FUNCTION_BLOCK FB_GameSetup
VAR_INPUT
END_VAR
VAR_OUTPUT
END_VAR
VAR
	i	: DINT;
	j	: DINT;
	k	: DINT;
	m	: INT;
END_VAR

// Decode sequencer step bits
MEMSET(ADR(GVL_Global.bStep), 0, SIZEOF(GVL_Global.bStep));
GVL_Global.stGameSetup.stStep[GVL_Global.stGameSetup.iStepNumber] := TRUE;

//Choose blackjack variation: 1 - Common BlackJack, 2 - Free Bet BlackJack, 3 - Spanish 21
IF GVL_Global.eBJVariation.Idle = GVL_Global.iVariationSelection THEN
	//Wait for user to select a BlackJack variation
	GVL_Global.sInstruction := 'Please choose a blackjack variation to play.';
END_IF

IF GVL_Global.iVariationSelection >= 1 AND GVL_Global.iVariationSelection <= 3 THEN
	//Set up initial information regarding card, card suit, and deck information
	FOR m := 0 TO 9 DO
		GVL_Global.stGameSetup.sCards[m] := INT_TO_STRING(m+2);
	END_FOR
	GVL_Global.stGameSetup.sCards[10] := 'J';
	GVL_Global.stGameSetup.sCards[11] := 'Q';
	GVL_Global.stGameSetup.sCards[12] := 'K';
	GVL_Global.stGameSetup.sCards[13] := 'A';
	
	GVL_Global.stGameSetup.sCardSuit[0] := 'Clubs';
	GVL_Global.stGameSetup.sCardSuit[1] := 'Diamonds';
	GVL_Global.stGameSetup.sCardSuit[2] := 'Bishops';
	GVL_Global.stGameSetup.sCardSuit[3] := 'Hearts';
	GVL_Global.stGameSetup.iStepNumber := 2;
ELSE
	GVL_Global.stGameSetup.iStepNumber := 0;
END_IF

//GVL_Global.sInstruction := 'Please choose a blackjack variation to play.';
//IF GVL_Global.iVariationSelection >=1 AND GVL_Global.iVariationSelection <= 3 THEN
//	GVL_Global.stGameSetup.iStepNumber := 2;
//ELSE
//	GVL_Global.stGameSetup.iStepNumber := 0;
//END_IF

//Error State
IF GVL_Global.stGameSetup.stStep.bStep[0] THEN
	//False entry was entered
	GVL_Global.stGamePlay.sMessageType.sErrorMessage := 'You entered a wrong variation input. Please try again.';
	GVL_Global.stGamePlay.bVariationSelected := FALSE;
	GVL_Global.stGamePlay.iVariationSelection := 0;
END_IF


//Idle State
IF GVL_Global.stGameSetup.stStep.bStep[1] THEN
	GVL_Global.stGamePlay.sMessageType.sErrorMessage := 'Game is ongoing.';
	IF GVL_Global.stGamePlay.bReadyToStart AND GVL_Global.stGameSetup.bBankRollComplete THEN
		GVL_Global.stGamePlay.iStepNumber := 1;
	ELSE
		GVL_Global.stGamePlay.iStepNumber := 0;
	END_IF
END_IF

//Blackjack Deviation Selection
IF GVL_Global.stGameSetup.stStep.bStep[2] THEN
	IF GVL_Global.eBJVariation.Common_BlackJack = GVL_Global.iVariationSelection THEN
		//Common Blackjack was selected
		GVL_Global.stGameSetup.stMessageType.sInstructionMessage := 'Variation selected: Common Blackjack.';
	ELSIF GVL_Global.eBJVariation.FreeBet_BlackJack = GVL_Global.iVariationSelection THEN
		GVL_Global.stGameSetup.stMessageType.sInstructionMessage := 'Variation selected: Free Bet Blackjack.';
	ELSIF GVL_Global.eBJVariation.Spanish21 = GVL_Global.iVariationSelection THEN
		GVL_Global.stGameSetup.stMessageType.sInstructionMessage := 'Variation selected: Spanish 21.';
	END_IF
	GVL_Global.stGameSetup.iStepNumber := 3;
END_IF

//Choose 2 sidebets: 1 - Buster BlackJack, 2 - Dealer 16, 3 - Lucky Lucky, 4 - Match the Dealer, 5 - Pot of Gold (TBD)
//Side Bets Selection
IF GVL_Global.stGameSetup.stStep.bStep[3] THEN
	GVL_Global.stGameSetup.stMessageType.sRulesForGame[0] := 'Choose two (2) side bets: 1 - Buster BlackJack, 2 - Dealer 16, 3 - Lucky Lucky, 4 - Match the Dealer, 5 - Pot of Gold';
	GVL_Global.stGameSetup.stMessageType.sInstructionMessage[1] := 'Enter in text box labeled -> Side Bets To Play';
	GVL_Global.stGameSetup.stMessageType.sInstructionMessage[2] := 'Choose two (2) side bets: 1 - Buster BlackJack, 2 - Dealer 16, 3 - Lucky Lucky, 4 - Match the Dealer, 5 - Pot of Gold';
	GVL_Global.stGameSetup.stMessageType.sInstructionMessage := 'Enter in the following prompt: #,#';
	//Side Bet Choices Decoded
	GVL_Global.stGameSetup.stSideBetChoice.iFind := FIND(',',GVL_Global.stGameSetup.stSideBetChoice.sSideBetSelections);
	GVL_Global.stGameSetup.stSideBetChoice.iSideBet_One := STRING_TO_INT(LEFT(GVL_Global.stGameSetup.stSideBetChoice.sSideBetSelections,GVL_Global.stGameSetup.stSideBetChoice.iFind-1));
	GVL_Global.stGameSetup.stSideBetChoice.iSideBet_Two := STRING_TO_INT(RIGHT(GVL_Global.stGameSetup.stSideBetChoice.sSideBetSelections,GVL_Global.stGameSetup.stSideBetChoice.iFind+1));
	//Side bet #1 chosen
	IF GVL_Global.stGameSetup.stSideBetChoice.iSideBet_One = GVL_Global.stGameSetup.stSideBetChoice.eSideBetChoice.BusterBlackjack THEN
		GVL_Global.stGameSetup.stSideBetChoice.bBusterBlackjackSelected := TRUE;
		//GVL_Global.stGameSetup.sSideBetChoice.iSideBetSelections.0 := TRUE;
	ELSIF GVL_Global.stGameSetup.stSideBetChoice.iSideBet_One = GVL_Global.stGameSetup.stSideBetChoice.eSideBetChoice.Dealer16 THEN
		GVL_Global.stGameSetup.stSideBetChoice.bDealer16Selected := TRUE;
		//GVL_Global.stGameSetup.sSideBetChoice.iSideBetSelections.1 := TRUE;
	ELSIF GVL_Global.stGameSetup.stSideBetChoice.iSideBet_One = GVL_Global.stGameSetup.stSideBetChoice.eSideBetChoice.LuckyLucky THEN
		GVL_Global.stGameSetup.stSideBetChoice.bLuckyLuckySelected := TRUE;
		//GVL_Global.stGameSetup.sSideBetChoice.iSideBetSelections.2 := TRUE;
	ELSIF GVL_Global.stGameSetup.stSideBetChoice.iSideBet_One = GVL_Global.stGameSetup.stSideBetChoice.eSideBetChoice.MatchtheDealer THEN
		GVL_Global.stGameSetup.stSideBetChoice.bMatchtheDealerSelected := TRUE;
	END_IF
	//Side bet #2 chosen
	IF GVL_Global.stGameSetup.stSideBetChoice.iSideBet_Two = GVL_Global.stGameSetup.stSideBetChoice.eSideBetChoice.BusterBlackjack THEN
		GVL_Global.stGameSetup.stSideBetChoice.bBusterBlackjackSelected := TRUE;
	ELSIF GVL_Global.stGameSetup.stSideBetChoice.iSideBet_Two = GVL_Global.stGameSetup.stSideBetChoice.eSideBetChoice.Dealer16 THEN
		GVL_Global.stGameSetup.stSideBetChoice.bDealer16Selected := TRUE;
	ELSIF GVL_Global.stGameSetup.stSideBetChoice.iSideBet_Two = GVL_Global.stGameSetup.stSideBetChoice.eSideBetChoice.LuckyLucky THEN
		GVL_Global.stGameSetup.stSideBetChoice.bLuckyLuckySelected := TRUE;
	ELSIF GVL_Global.stGameSetup.stSideBetChoice.iSideBet_Two = GVL_Global.stGameSetup.stSideBetChoice.eSideBetChoice.MatchtheDealer THEN
		GVL_Global.stGameSetup.stSideBetChoice.bMatchtheDealerSelected := TRUE;
	END_IF
	
	IF GVL_Global.stGameSetup.stSideBetChoice.iSideBet_One <> 0 AND GVL_Global.stGameSetup.stSideBetChoice.iSideBet_Two <> 0 THEN
		GVL_Global.stGameSetup.iStepNumber := 4;
	END_IF
END_IF

//Input number of players/hands to be dealt. Max of 6.
IF GVL_Global.stGameSetup.stStep.bStep[4] THEN
	GVL_Global.stGamePlay.sMessageType.sInstructionMessage := 'Please enter number of players/hands going to play';
	IF GVL_Global.stTable.iNumberofPlayers >= 1 AND GVL_Global.stTable.iNumberofPlayers <= 6 THEN
		//GVL_Global.stTable.iNumberofPlayers;
		FOR i := 1 TO GVL_Global.stTable.iNumberofPlayers DO
			GVL_Global.stGameSetup.stPlayer[i].bSeatPlaying := TRUE;	
		END_FOR
		//GVL_Global.stGameSetup.iSeatsOpen := GVL_Global.stTable.iNumberofPlayers + 1;
		GVL_Global.stGamePlay.iStepNumber := 5;
	ELSE
		//Number of players entered is invalid.
		GVL_Global.stGameSetup.stMessageType.sErrorMessage := 'Entered invalid number of players. Please try again.';
	END_IF
	//
//GVL_Global.stGamePlay.iStepNumber := 3;
END_IF

//Input number of decks to be dealt.
IF GVL_Global.stGameSetup.stStep.bStep[5] THEN
	GVL_Global.stGamePlay.sMessageType.sInstructionMessage := 'Please enter number of decks to deal (1-6)';
	IF GVL_Global.stTable.iNumberofDecks >= 1 AND GVL_Global.stTable.iNumberofDecks <= 6 THEN
		GVL_Global.stGamePlay.sMessageType.sInstructionMessage := CONCAT('Dealer will deal a total of ',DINT_TO_STRING(GVL_Global.stTable.iNumberofDecks));
		GVL_Global.stGamePlay.iStepNumber := 6;
	ELSE
		//Number of decks entered is invalid.
		GVL_Global.stGameSetup.stMessageType.sErrorMessage := 'Entered invalid number of decks. Please try again.';
	END_IF
END_IF

//Input table minimum bet.
IF GVL_Global.stGameSetup.stStep.bStep[6] THEN
	GVL_Global.stGamePlay.sMessageType.sInstructionMessage := 'Please enter the minimum bet to play.';
	IF GVL_Global.stTable.iMinimumBet >= 5 THEN
		GVL_Global.stGamePlay.sMessageType.sInstructionMessage := CONCAT('Minimum table bet is ',DINT_TO_STRING(GVL_Global.stTable.iMinimumBet));
		GVL_Global.stGamePlay.iStepNumber := 7;
	ELSE
		//Number of decks entered is invalid.
		GVL_Global.stGameSetup.stMessageType.sErrorMessage := 'Entered an invalid table bet. Please try again.';
	END_IF
END_IF

//Input table max bet. - May not use - TBD
IF GVL_Global.stGameSetup.stStep.bStep[7] THEN
	GVL_Global.stGamePlay.iStepNumber := 8;
END_IF

//Set up players/seats who are playing.
IF GVL_Global.stGameSetup.stStep.bStep[8] THEN
	FOR j := 1 TO GVL_Global.stTable.iNumberofPlayers DO
		GVL_Global.stGameSetup.stPlayer[j].iSeat := j;
	END_FOR
	GVL_Global.stGamePlay.iStepNumber := 9;
END_IF

//Input starting bank roll.
IF GVL_Global.stGameSetup.stStep.bStep[9] THEN
	GVL_Global.stGamePlay.sMessageType.sInstructionMessage := 'Please enter bankroll for each player.';
	IF GVL_Global.stGameSetup.bBankRollComplete THEN
		GVL_Global.stGamePlay.sMessageType := 'Details for chips: Reds - 5, Whites - 25, Blues - 100, Greens - 500, Blacks - 1 or 1000';
		GVL_Global.stGamePlay.iStepNumber := 10;
	END_IF
END_IF

//Chips given: Reds - $5, Whites - $25, Blues - $100, Greens - $500, Blacks - $1  

//Finalize Game Setup
IF GVL_Global.stGameSetup.stStep.bStep[10] THEN
	GVL_Global.stGamePlay.sMessageType.sInstructionMessage := 'Ready to start the game?';
	IF GVL_Global.stGamePlay.bReadyToStart THEN
		GVL_Global.stGameSetup.bGameSetupComplete := TRUE;
		GVL_Global.stGamePlay.iStepNumber := 1;
	END_IF
END_IF

END_FUNCTION_BLOCK

(* stored: Version 1.1.0.1, ProductVersion 3.1.4024.10
   POU FB_GameSetup: Id {84ee8ec1-a4ad-4f71-bbc3-2b9c2539696b}, SpecialFunc None *)
